Staubli VAL3: Control_PatMove.pgx

public program Control_PatMove(num& x_nStart, num& x_nEnd)
  local string l_sItem[6]
  local num l_nNum
  local num l_nKey
  local num l_nData[6]
  local num l_nSelectIndex
begin
  //为LasMAN3.7进行配置
  //中途进行模拟点

  l_nData[0]=x_nStart
  l_nData[1]=x_nEnd


  l_sItem[0]="开始模拟点:"+toString(".3",l_nData[0])
  l_sItem[1]="结束模拟点:"+toString(".3",l_nData[1])


  call Control_BottomS(",,,,,,,确定")
  call Control_PanelXY(8,0,15,2)
  call Control_Panel("切割点局部模拟")
  call Control_List(l_sItem,l_nSelectIndex)
  while true
    l_nKey=getKey()

    switch l_nKey
      case 261
        l_nSelectIndex=max(0,l_nSelectIndex-1)
      break

      case 266
        l_nSelectIndex=min(l_nSelectIndex+1,1)
      break

      case 278
        x_nStart=l_nData[0]
        x_nEnd=l_nData[1]
        cls()
        return
      break


      //      case 277,255
      //
      //        cls()
      //        return
      //      break

      case 270
        call Float_Edit(l_nData[l_nSelectIndex],nPanelLTopX+12,l_nSelectIndex+nPanelLTopY+1)
      break

    endSwitch

    if l_nKey!=-1
      l_sItem[0]="开始模拟点:"+toString(".3",l_nData[0])
      l_sItem[1]="结束模拟点:"+toString(".3",l_nData[1])

      call Control_List(l_sItem,l_nSelectIndex)

    endIf






  endWhile





end
